TYPE ST_GZ_DLK_Zustand :
STRUCT
	Freigabe			: BOOL;
	Blindleistung		: REAL;		(*Wert des Universalmessgerätes UMG604*)
	Blindarbeit			: REAL;		(*Wert des Universalmessgerätes UMG604*)
	Scheinleistung		: REAL;		(*Wert des Universalmessgerätes UMG604*)
	Scheinarbeit		: REAL;		(*Wert des Universalmessgerätes UMG604*)
	Wirkleistung		: REAL;		(*Wert des Universalmessgerätes UMG604*)
	Wirkarbeit			: REAL;		(*Wert des Universalmessgerätes UMG604*)
	Zaehler_Hauptanschluss_Volumen	: REAL;		(*Wert des Universalmessgerätes UMG604*)
END_STRUCT
END_TYPE

(* stored: Version 1.1.0.1, ProductVersion 3.1.4024.9
   DUT ST_GZ_DLK_Zustand: Id {86d300c5-65d1-41c2-bd59-5b49a41eaccb} *)
